FUNCTION WRITE_ANY_SINT : BOOL
VAR_INPUT
    ptr: POINTER TO SINT;
    val: SINT;
END_VAR

ptr^ := val;

END_FUNCTION

(* stored: Version 1.1.0.1, ProductVersion 3.1.4022.9
   POU WRITE_ANY_SINT: Id {e310eaa9-3123-4344-b07c-fc54b5c8e3ac}, SpecialFunc None *)
